FUNCTION TFAsseInFinestra : bool //Valuta se l'asse è nella finsetra di posizione desiderata
VAR_INPUT
	Posizione_Attuale 	: LREAL;
	Posizione_Finale 	: LREAL;
	FinestraDiControllo : REAL;
END_VAR
VAR
END_VAR

TFAsseInFinestra := FALSE;

IF Posizione_Attuale >= (Posizione_Finale - FinestraDiControllo/2) AND Posizione_Attuale <= (Posizione_Finale + FinestraDiControllo/2) THEN
	TFAsseInFinestra := TRUE;
	RETURN;
END_IF

END_FUNCTION

(* stored: Version 1.1.0.1, ProductVersion 3.1.4024.11
   POU TFAsseInFinestra: Id {05f046ad-1ef9-45bb-b233-5e93be03afd0}, SpecialFunc None *)
